Staubli VAL3: AA_Chessie.pjx

--- AA_Chessie.pjx ---
Parameters version=s7.9 stackSize=5000 millimeterUnit=true
Program file=CasesNoires.pgx
Program file=DeplacementInit.pgx
Program file=Deplacementpion.pgx
Program file=start.pgx
Program file=stop.pgx
Program file=TestPositionCal.pgx
Data file=AA_Chessie.dtx

--- AA_Chessie.dtx ---
jointRx jStart = {j1=-4.35, j2=22.39, j3=131, j5=25.77, j6=50.65}
jointRx jDepart = {j1=20.811233, j2=126.617326, j3=-10.855704, j5=64.238378, j6=-69.188767}
frame fFrame = {x=374.8, y=3.07, z=-517.036829, rx=-180, fatherId=world[0]}
pointRx pTable = {fatherId=fFrame[0]}
pointRx pCaseNoire[33]
  [0] = {x=374.8, y=3.07, z=-517.036829, rx=-180, shoulder=lefty, elbow=epositive, wrist=wpositive, fatherId=world[0]}
  [1] = {fatherId=world[0]}
  [2] = {fatherId=world[0]}
  [3] = {fatherId=world[0]}
  [4] = {fatherId=world[0]}
  [5] = {fatherId=world[0]}
  [6] = {fatherId=world[0]}
  [7] = {fatherId=world[0]}
  [8] = {fatherId=world[0]}
  [9] = {fatherId=world[0]}
  [10] = {fatherId=world[0]}
  [11] = {fatherId=world[0]}
  [12] = {fatherId=world[0]}
  [13] = {fatherId=world[0]}
  [14] = {fatherId=world[0]}
  [15] = {fatherId=world[0]}
  [16] = {fatherId=world[0]}
  [17] = {fatherId=world[0]}
  [18] = {fatherId=world[0]}
  [19] = {fatherId=world[0]}
  [20] = {fatherId=world[0]}
  [21] = {fatherId=world[0]}
  [22] = {fatherId=world[0]}
  [23] = {fatherId=world[0]}
  [24] = {fatherId=world[0]}
  [25] = {fatherId=world[0]}
  [26] = {fatherId=world[0]}
  [27] = {fatherId=world[0]}
  [28] = {fatherId=world[0]}
  [29] = {fatherId=world[0]}
  [30] = {fatherId=world[0]}
  [31] = {fatherId=world[0]}
  [32] = {fatherId=world[0]}
jointRx jCaseNoire = {j1=-7.236149, j2=83.896154, j3=110.243942, j5=-14.140096, j6=172.763851}
num nX
num nY
num ni
mdesc mPrise = {accel=25}
mdesc mDepose = {accel=25}
mdesc mDeplacement = {accel=250}
tool tTool = {x=2.67332365613152, y=0.0823457375943404, z=50.1043771229301, rx=-7.34240987449236E-12, ry=-8.49495425328202E-12, rz=2.13111140704977E-13, fatherId=flange[0], ioLink=valve1}
jointRx jInitial
trsf trAppro = {z=-10}

--- start.pgx ---
public program start()
begin
  // Position des cases
  //   28   29  30  31             ligne 8
  //     ....                      ...
  //  8   9  10  11                ligne 3
  //    4   5   6   7              ligne 2
  //  0   1   2   3                ligne 1
  //pCase[0] = case O en bas à gauche du plateau


  //se met en position 0
  call DeplacementInit()

  //Deplacementpion(X,Y) -> deplacement du pion de X vers Y
  call Deplacementpion(0,4)
  call Deplacementpion(4,5)
  call Deplacementpion(5,6)
  call Deplacementpion(6,7)
  call Deplacementpion(7,8)
  call Deplacementpion(8,31)




end

--- CasesNoires.pgx ---
public program CasesNoires()
begin


  // Position des cases
  //   28   29  30  31             ligne 8
  //     ....                      ...
  //  8   9  10  11                ligne 3
  //    4   5   6   7              ligne 2
  //  0   1   2   3                ligne 1

  //pCase[0] = case O en bas à gauche du plateau

  //variable pour numeroter les cases
  ni=0

  for nY=1 to 8
    for nX=0 to 3

      //ligne case impair
      if nY % 2 == 1
        pCaseNoire[ni]= compose(pCaseNoire[0], fFrame , {55.6*nX, -27.8*(nY - 1), 0, 0, 0, 0})
        //pCaseNoire[ni]= pCaseNoire[0] + 55.6*nX + 27.8 * (nY - 1)

      //ligne case pair
      else
        pCaseNoire[ni]= compose(pCaseNoire[0], fFrame , {27.8*(nX+1) + 27.8*nX, -27.8*(nY - 1), 0, 0, 0, 0})
        //pCaseNoire[ni]= pCaseNoire[0] + 27.8*(nX+1) + 27.8 * (nY - 1)
      endIf

      ni = ni + 1

    endFor
  endFor


end

--- DeplacementInit.pgx ---
program DeplacementInit()
begin
  movej(jInitial, tTool, mDeplacement)
end

--- Deplacementpion.pgx ---
public program Deplacementpion(num x_nPointDepart, num x_nPointArrivee)
begin
  //met à jour position des cases noires
  call CasesNoires()


  //Deplacementpion(X,Y) -> deplacement du pion de X vers Y


  //Deplacement vers le pion en X
  movej( appro(pCaseNoire[x_nPointDepart], trAppro), tTool, mDeplacement)

  //s'approche et prend le pion en X
  close(tTool)
  movel( pCaseNoire[x_nPointDepart], tTool, mPrise)
  open(tTool)

  movel( appro(pCaseNoire[x_nPointDepart], trAppro), tTool, mDeplacement)

  //Deplacement vers Y puis approche vers Y
  movej ( appro(pCaseNoire[x_nPointArrivee], trAppro), tTool, mDeplacement)
  movel( pCaseNoire[x_nPointArrivee], tTool, mPrise)

  //lache la piece et remonte
  close(tTool)
  movel( appro(pCaseNoire[x_nPointArrivee], trAppro), tTool, mDeplacement)


end

--- TestPositionCal.pgx ---
program TestPositionCal()
begin
  call DeplacementInit()

  call Deplacementpion(0,1)
  call Deplacementpion(31,30)
end
